KUKA KRL data list: Points.dat

&ACCESS RVP
DEFDAT Points
;FOLD EXTERNAL DECLARATIONS;%{PE}%MKUKATPBASIS,%CEXT,%VCOMMON,%P
;FOLD BASISTECH EXT;%{PE}%MKUKATPBASIS,%CEXT,%VEXT,%P
EXT  BAS (BAS_COMMAND  :IN,REAL  :IN )

DECL INT XTOOLBASE = 1
DECL INT XTOOL = 2

;ENDFOLD (BASISTECH EXT)
;FOLD USER EXT;%{E}%MKUKATPUSER,%CEXT,%VEXT,%P
;Make your modifications here

; =============================== ;
; Declaração de variáveis Globais ;
; =============================== ;

DECL POS PontoRecolhaArray[3]
DECL POS PontoDepositoArray[3]
DECL POS PontoIntermedioArray[6]

DECL INT count[3]; índices: 1=Amarelo, 2=Azul, 3=Verde

; ============================== ;
; Definição dos Inputs e Outputs ;
; ============================== ;
SIGNAL B_Branco $IN[20]
SIGNAL B_VERMELHO $IN[21]
SIGNAL B_PRETO $IN[22]

SIGNAL IN_POS1_AMARELO $IN[11]
SIGNAL IN_POS1_AZUL    $IN[12]
SIGNAL IN_POS1_VERDE   $IN[13]

SIGNAL IN_POS2_AMARELO $IN[14]
SIGNAL IN_POS2_AZUL    $IN[15]
SIGNAL IN_POS2_VERDE   $IN[16]

SIGNAL IN_POS3_AMARELO $IN[17]
SIGNAL IN_POS3_AZUL    $IN[18]
SIGNAL IN_POS3_VERDE   $IN[19]

SIGNAL LARANJA $OUT[23]
SIGNAL VERDE $OUT[22]
SIGNAL AZUL $OUT[21]
; ============================== ;
; Posição Inicial
DECL POS HOME = {X 200, Y 376.5, Z -147, C 0} ; HOME

; Posições de Recolha
DECL POS P1_Recolha = {X 65.5, Y 224, Z -140, C 24}   ; P1
DECL POS P2_Recolha = {X 64.5, Y 152.5, Z -140, C 24} ; P2
DECL POS P3_Recolha = {X 53.5, Y 82, Z -140, C 24}    ; P3

; Posições de Depósito
DECL POS P1_Deposito = {X 353, Y 299, Z -140, C 2.5}  ; Azul (Junto)
DECL POS P2_Deposito = {X 268, Y 299, Z -140, C 2.5}  ; Amarelo (Meio)
DECL POS P3_Deposito = {X 184, Y 299, Z -140, C 2.5}  ; Verde (Fundo)

; Posições Intermédias
DECL POS P1_Intermedia = {X 65.5, Y 224, Z -80, C 84}    ;P1
DECL POS P2_Intermedia = {X 64.5, Y 152.5, Z -80, C 84}  ;P2
DECL POS P3_Intermedia = {X 53.5, Y 82, Z -80, C 84}     ;P3
DECL POS P4_Intermedia = {X 688, Y 234, Z -80, C 0}      ; Azul
DECL POS P5_Intermedia = {X 688, Y 145, Z -80, C 0}      ; Amarelo
DECL POS P6_Intermedia = {X 688, Y 64, Z -80, C 0}       ; Verde


;ENDFOLD (USER EXT)
;ENDFOLD (EXTERNAL DECLARATIONS)
DECL PDAT PDAT1 = {APO_MODE #CDIS, APO_DIST 500, VEL 80, ACC 80, GEAR_JERK 100.0, EXAX_IGN 0}
DECL PDAT PDAT2 = {APO_MODE #CDIS, APO_DIST 10, VEL 60, ACC 30, GEAR_JERK 100.0, EXAX_IGN 0}
DECL PDAT PDAT3 = {APO_MODE #CDIS, APO_DIST 500, VEL 80, ACC 80, GEAR_JERK 100.0, EXAX_IGN 0}
DECL PDAT PDAT4 = {APO_MODE #CDIS, APO_DIST 10, VEL 60, ACC 30, GEAR_JERK 100.0, EXAX_IGN 0}
DECL PDAT PDAT5 = {APO_MODE #CDIS, APO_DIST 500, VEL 80, ACC 80, GEAR_JERK 100.0, EXAX_IGN 0}
DECL PDAT PDAT6 = {APO_MODE #CDIS, APO_DIST 10, VEL 60, ACC 30, GEAR_JERK 100.0, EXAX_IGN 0}
DECL PDAT PDAT7 = {APO_MODE #CDIS, APO_DIST 500, VEL 80, ACC 80, GEAR_JERK 100.0, EXAX_IGN 0}
DECL PDAT PDAT8 = {APO_MODE #CDIS, APO_DIST 10, VEL 60, ACC 30, GEAR_JERK 100.0, EXAX_IGN 0}
DECL PDAT PDAT9 = {APO_MODE #CDIS, APO_DIST 500, VEL 80, ACC 80, GEAR_JERK 100.0, EXAX_IGN 0}
DECL PDAT PDAT10 = {APO_MODE #CDIS, APO_DIST 10, VEL 60, ACC 30, GEAR_JERK 100.0, EXAX_IGN 0}

ENDDAT
